FUNCTION_BLOCK XtsEnableSequence  IMPLEMENTS I_Task
VAR
	_caGroup : I_CollisionGroup;
	moverIndex : UINT;
	AllMoversEnabled: BOOL;
	EnableTrigger : BOOL;	
	arrMovers : ARRAY[0..MaxMovers] OF I_XtsMover;
	_registeredNumberOfMovers : INT;
	State: EnableState;
	_Done: BOOL;
	_Error: BOOL;
	_Busy: BOOL;
END_VAR
VAR CONSTANT
	MaxMovers : INT := 255;
END_VAR

{analysis -2}

METHOD Abort : BOOL
EnableTrigger := FALSE;
State := 0;
END_METHOD

PROPERTY Busy : BOOL
GET
Busy := _Busy;
END_GET
END_PROPERTY

METHOD Cycle : HRESULT
VAR
	i : INT;
END_VAR
CASE State OF
	EnableState.Idle:
		IF EnableTrigger THEN
			Cycle := S_PENDING;
			State := EnableState.Reset_Movers;
			EnableTrigger := FALSE;
			moverIndex := 0;
			_Busy := TRUE;
			_Done := FALSE;
			_Error := FALSE;
		END_IF
		
	EnableState.Reset_Movers:
		FOR i := 0 TO (_registeredNumberOfMovers-1) DO
			arrMovers[i].Reset();
		END_FOR
		State := EnableState.Reset_Group;
		
	EnableState.Reset_Group:
		IF _caGroup.IsInErrorStop THEN
			_caGroup.Reset();
		END_IF
		State := EnableState.Add_Mover;
		
	EnableState.Add_Mover:
		IF Succeeded( _caGroup.AddMoverToThisGroup(MoverToAdd := arrMovers[moverIndex])) THEN
			State := EnableState.Check_Add_Mover;
		END_IF
		
		
	EnableState.Check_Add_Mover:
		IF moverIndex <> (_registeredNumberOfMovers-1) THEN
			moverIndex := moverIndex + 1;
			State := EnableState.Add_Mover;
		ELSE
			FOR i := 0 TO (_registeredNumberOfMovers-1) DO
				arrMovers[i].EnableMover();
			END_FOR
			State := EnableState.Enable_Movers;
		END_IF
		
	EnableState.Enable_Movers:
		AllMoversEnabled := TRUE;
		FOR i := 0 TO (_registeredNumberOfMovers-1) DO
			AllMoversEnabled := TRUE AND arrMovers[i].IsEnabled;
		END_FOR
		IF AllMoversEnabled THEN
			
			State := EnableState.Enable_Group;
		END_IF

	EnableState.Enable_Group:
		IF _caGroup.Enable() THEN
			State := EnableState.Check_Standby;
		END_IF
		
	EnableState.Check_Standby:
		IF _caGroup.IsInStandBy THEN
			State := EnableState.Idle;
			_Busy := FALSE;
			_Done := TRUE;
			Cycle := S_OK;
		END_IF
	ELSE
		Cycle := E_FAIL;
		_Busy := FALSE;
		_Done := FALSE;
		_Error := TRUE;
END_CASE
END_METHOD

PROPERTY Done : BOOL
GET
Done := _Done;
END_GET
END_PROPERTY

METHOD Enable : HRESULT
VAR_INPUT
END_VAR
IF _Busy THEN
	Enable := -1;
	RETURN;
END_IF

IF EnableTrigger THEN
	Enable := -2;
	RETURN;
END_IF

IF _caGroup = 0 THEN
	Enable := -3;
	RETURN;
END_IF

EnableTrigger := TRUE;
END_METHOD

PROPERTY Error : BOOL
GET
Error := _Error;
END_GET
END_PROPERTY

PROPERTY MyCollisionGroup : I_CollisionGroup
GET
MyCollisionGroup := _caGroup;
END_GET
SET
_caGroup := MyCollisionGroup;
END_SET
END_PROPERTY

METHOD RegisterMovers : HRESULT
VAR_INPUT
	MyMover : I_XtsMover;
END_VAR
arrMovers[_registeredNumberOfMovers] := MyMover;
_registeredNumberOfMovers := _registeredNumberOfMovers + 1;
END_METHOD

END_FUNCTION_BLOCK

(* stored: Version 1.1.0.1
   POU XtsEnableSequence: Id {b7e7ab09-3a30-4ddb-a242-e0b5aa00cbc9}, SpecialFunc None
   Method Abort: Id {9cec9788-9ce4-4a9f-821c-172bdb3141aa}
   Property Busy: Id {bc4497ef-9c3a-4d02-9785-8733db6c9845}
   Get Get: Id {d45d9021-7bdc-468f-89fe-ec603e3e38b0}
   Method Cycle: Id {2913b891-dfae-43d9-b9d3-4a1a1101f452}
   Property Done: Id {81ec7814-89cb-4301-940b-bd26fe7c0dd9}
   Get Get: Id {f5e4b06f-0267-4980-bd12-ca8f03d203a3}
   Method Enable: Id {1c2a3468-bb52-4165-8d13-732b960a1dd0}
   Property Error: Id {de4172ae-7561-44d0-9211-14ccf56f7fba}
   Get Get: Id {7981ac0e-81ff-46ad-91e6-7e6c0cd85d62}
   Property MyCollisionGroup: Id {0c241349-a398-40a0-a115-326a5cd04bf6}
   Get Get: Id {c45de961-c00e-41dd-bc0b-0921ea45f3ce}
   Set Set: Id {0715b558-a706-48d8-a891-3862516fa554}
   Method RegisterMovers: Id {330a136c-c434-49ce-bb82-6de99c18307c} *)
